{attribute 'linkalways'} 
{attribute 'no_explicit_call' := 'This FB is a CLASS and must be accessed using methods or properties'}
{attribute 'enable_dynamic_creation'}
FUNCTION_BLOCK Node_F_VN_MinElementElementwise_TcVnVector3_UINT EXTENDS VisionNode
VAR
    ipContainer : _ITcVnContainer;
    aMin : _TcVnVector3_UINT;
    hrPrev : _HRESULT(S_OK);
    hresult : _HRESULT(S_OK);
END_VAR

METHOD PUBLIC  Clone : I_Node
VAR
	pNode : POINTER TO Node_F_VN_MinElementElementwise_TcVnVector3_UINT;
END_VAR
pNode := __NEW(Node_F_VN_MinElementElementwise_TcVnVector3_UINT);
Clone := pNode^;
END_METHOD

METHOD FB_init : BOOL
VAR_INPUT
	bInitRetains : BOOL; // if TRUE, the retain variables are initialized (warm start / cold start)
	bInCopyCode : BOOL;  // if TRUE, the instance afterwards gets moved into the copy code (online change)
END_VAR
AddInput('ipContainer', ipContainer);
AddInput('hrPrev', hrPrev);
AddOutput('ipContainer', ipContainer);
AddOutput('aMin', aMin);
AddOutput('hresult',hresult);
END_METHOD

METHOD PROTECTED OnExecute
hresult.Value := F_VN_MinElementElementwise_TcVnVector3_UINT(
    ipContainer := ipContainer.Value,
    aMin := aMin.Value,
    hrPrev:= hrPrev.Value);
END_METHOD

METHOD PUBLIC PreExecutionCheck
VAR_INPUT
	Check : I_PreExecutionChecks;
END_VAR
Check.IsTrue(ipContainer.IsValid, 'ipContainer must be a valid container');
Check.IsTrue(ipContainer.IsType(TC_GLOBAL_CONST_LIST.ContainerType_Vector_TcVnVector3_UINT), 'ipContainer contains incorrect type');
END_METHOD

END_FUNCTION_BLOCK

(* stored: Version 1.1.0.1, ProductVersion 3.1.4026.13
   POU Node_F_VN_MinElementElementwise_TcVnVector3_UINT: Id {1f304089-662d-4c0c-b96d-a1989ff582ea}, SpecialFunc None
   Folder Constructor: Id {54afa2e6-2368-457e-a8e4-39cc59c3f98e}
   Method Clone: Id {8219cf20-f251-4b2f-80bc-bb896ec47354}
   Method FB_init: Id {05305b98-3291-4c60-8b16-9ea9ecce2490}
   Method OnExecute: Id {70df69a8-3e05-4a59-9f7b-4ab4984fab35}
   Method PreExecutionCheck: Id {64308ae0-36cb-4e9d-8104-6b8c998a3eb5} *)
